TYPE T_TCP_RT_CLIENT_CTRL :
STRUCT
	bExecute: 	BOOL 	:= FALSE;
	sCmd:		STRING;
END_STRUCT
END_TYPE

(* stored: Version 1.1.0.1, ProductVersion 3.1.4022.16
   DUT T_TCP_RT_CLIENT_CTRL: Id {14882210-ac57-46db-b880-7468f9d13bae} *)
